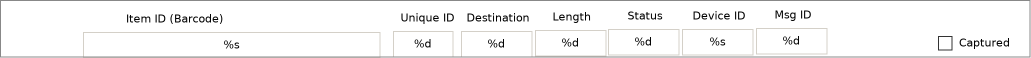
VISUALIZATION ArrayInspection  // 1031x58
VAR_IN_OUT
	st_ItemExt_Disp	:		ST_ItemExt;
(*	ID : STRING := '';		// Bar Code 	
	UniqueID : DINT := 0;		// Generic ID for tracking
	Destination : DINT := 0;
	Length : DINT := 0;
	Status : E_StatusCode := E_StatusCode.No_Status;
	CapturedInMetrics : BOOL;
	DeviceID:	STRING(5);	// Device ID associated with this record
	MessageType:	E_MessageIds;	// Message Type associated with this record
E*)
END_VAR
    Textfield (83,32 297x26), "%s", text variable: st_ItemExt_Disp.ID
    Label (86,11 178x16), "Item ID (Barcode)", invisible if: D
    Label (396,10 63x16), "Unique ID", invisible if: D
    Textfield (393,31 60x26), "%d", text variable: st_ItemExt_Disp.UniqueID
    Label (464,10 68x16), "Destination", invisible if: D
    Textfield (461,31 71x26), "%d", text variable: st_ItemExt_Disp.Destination
    Label (538,9 68x16), "Length", invisible if: D
    Textfield (535,30 71x26), "%d", text variable: st_ItemExt_Disp.Length
    Label (611,8 68x16), "Status", invisible if: D
    Textfield (608,29 71x26), "%d", text variable: st_ItemExt_Disp.Status
    Checkbox (936,28 95x30), "Captured", variable: st_ItemExt_Disp.CapturedInMetrics
    Textfield (682,29 71x26), "%s", text variable: st_ItemExt_Disp.DeviceID
    Label (685,8 68x16), "Device ID", invisible if: D
    Textfield (756,28 71x26), "%d", text variable: st_ItemExt_Disp.MessageType
    Label (759,7 68x16), "Msg ID", invisible if: D
END_VISUALIZATION

(* stored: Version 1.1.0.1, ProductVersion 3.1.4024.4
   Visu ArrayInspection: Id {d55ba907-b0ad-468b-9509-b3bea94354d3} *)
